PROGRAM PulsGenerator
VAR
	fbBlinking,fbBlinking1,fbBlinking2,fbBlinking3,fbBlinking4,fbBlinking5		:FB_Blinking;
	pPulsOutput			:POINTER TO S_PlusOutput;
	
END_VAR

pPulsOutput := ADR(GVL_General.PlusOutput);


fbBlinking(pVariable:= ADR(pPulsOutput^.Puls100ms) , interval:= T#100MS);

fbBlinking1(pVariable:= ADR(pPulsOutput^.Puls1s) , interval:= T#1S);

fbBlinking2(pVariable:= ADR(pPulsOutput^.Puls200ms) , interval:= T#200MS);

fbBlinking3(pVariable:= ADR(pPulsOutput^.Puls2s) , interval:= T#2S);

fbBlinking4(pVariable:= ADR(pPulsOutput^.Puls500ms) , interval:= T#500MS);

fbBlinking5(pVariable:= ADR(pPulsOutput^.Puls800ms) , interval:= T#800MS);

END_PROGRAM

(* stored: Version 1.1.0.1, ProductVersion 3.1.4022.16
   POU PulsGenerator: Id {09f64a5a-bb1b-444d-a8a2-59f66c7db939}, SpecialFunc None *)
